SUBAPPLICATION ACTION_CLIENT_STATUS
  (* Standard: 61499-2 *)
  (* Version 1.0, 2023-03-23, Tim Hesse *)
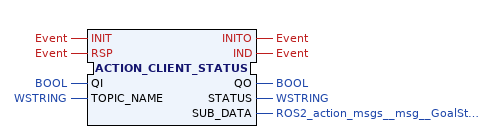
  EVENT_INPUT
    INIT; (* Initialization Request *)
    RSP;
  END_EVENT
  EVENT_OUTPUT
    INITO; (* Initialization Confirm *)
    IND;
  END_EVENT
  VAR_INPUT
    QI : BOOL; (* Input event qualifier *)
    TOPIC_NAME : WSTRING;
  END_VAR
  VAR_OUTPUT
    QO : BOOL; (* Output event qualifier *)
    STATUS : WSTRING;
    SUB_DATA : ROS2_action_msgs__msg__GoalStatusArray;
  END_VAR
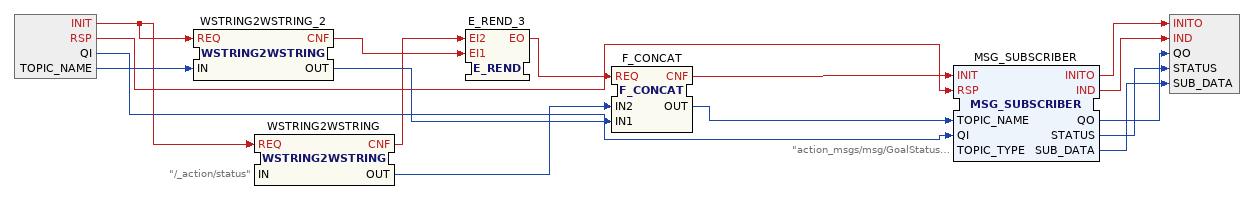
  FBS
    WSTRING2WSTRING_2 : WSTRING2WSTRING;
    F_CONCAT : F_CONCAT;
    E_REND_3 : E_REND;
    WSTRING2WSTRING : WSTRING2WSTRING(IN := "/_action/status");
  END_FBS
  SUBAPPS
    MSG_SUBSCRIBER : MSG_SUBSCRIBER(TOPIC_TYPE := "action_msgs/msg/GoalStatusArray");
  END_SUBAPPS
  EVENT_CONNECTIONS
    WSTRING2WSTRING.CNF TO E_REND_3.EI2;
    E_REND_3.EO TO F_CONCAT.REQ;
    WSTRING2WSTRING_2.CNF TO E_REND_3.EI1;
    F_CONCAT.CNF TO MSG_SUBSCRIBER.INIT;
    INIT TO WSTRING2WSTRING_2.REQ;
    RSP TO MSG_SUBSCRIBER.RSP;
    INIT TO WSTRING2WSTRING.REQ;
    MSG_SUBSCRIBER.INITO TO INITO;
    MSG_SUBSCRIBER.IND TO IND;
  END_CONNECTIONS
  DATA_CONNECTIONS
    F_CONCAT.OUT TO MSG_SUBSCRIBER.TOPIC_NAME;
    WSTRING2WSTRING.OUT TO F_CONCAT.IN2;
    WSTRING2WSTRING_2.OUT TO F_CONCAT.IN1;
    QI TO MSG_SUBSCRIBER.QI;
    TOPIC_NAME TO WSTRING2WSTRING_2.IN;
    MSG_SUBSCRIBER.QO TO QO;
    MSG_SUBSCRIBER.STATUS TO STATUS;
    MSG_SUBSCRIBER.SUB_DATA TO SUB_DATA;
  END_CONNECTIONS
END_SUBAPPLICATION
